FUNCTION_BLOCK BatteryModelServer (* Client FB for delegating battery model simulations to an external client. *)
  (* Standard: 61499-2 *)
  (* Version 1.0, 2017-06-18, Marc Jakobi, HTW Berlin *)
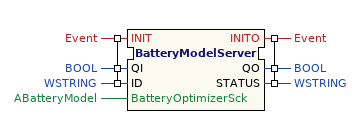
  EVENT_INPUT
    INIT WITH QI, ID; (* Initialization Request *)
  END_EVENT
  EVENT_OUTPUT
    INITO WITH QO, STATUS; (* Initialization Confirm *)
  END_EVENT
  VAR_INPUT
    QI : BOOL; (* Input event qualifier *)
    ID : WSTRING; (* Connection Identifier *)
  END_VAR
  VAR_OUTPUT
    QO : BOOL; (* Output event qualifier *)
    STATUS : WSTRING; (* Service Status *)
  END_VAR
  SOCKETS
    BatteryOptimizerSck : ABatteryModel; (* Link to BatteryOptimizer *)
  END_SOCKETS
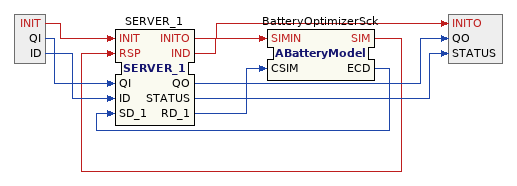
  FBS
    SERVER_1 : SERVER_1;
  END_FBS
  EVENT_CONNECTIONS
    INIT TO SERVER_1.INIT;
    SERVER_1.INITO TO INITO;
    SERVER_1.IND TO BatteryOptimizerSck.SIMIN;
    BatteryOptimizerSck.SIM TO SERVER_1.RSP;
  END_CONNECTIONS
  DATA_CONNECTIONS
    QI TO SERVER_1.QI;
    ID TO SERVER_1.ID;
    BatteryOptimizerSck.ECD TO SERVER_1.SD_1;
    SERVER_1.QO TO QO;
    SERVER_1.STATUS TO STATUS;
    SERVER_1.RD_1 TO BatteryOptimizerSck.CSIM;
  END_CONNECTIONS
END_FUNCTION_BLOCK
